// LS Electric XG5000 project: 동남138
// PLC NewPLC
// module base 0 slot 0: 입출력 모듈:XBC-DN/DP14E (DC 24V 입력 8점, 트랜지스터 출력 6점)

PROGRAM NewProgram (task: 스캔 프로그램)

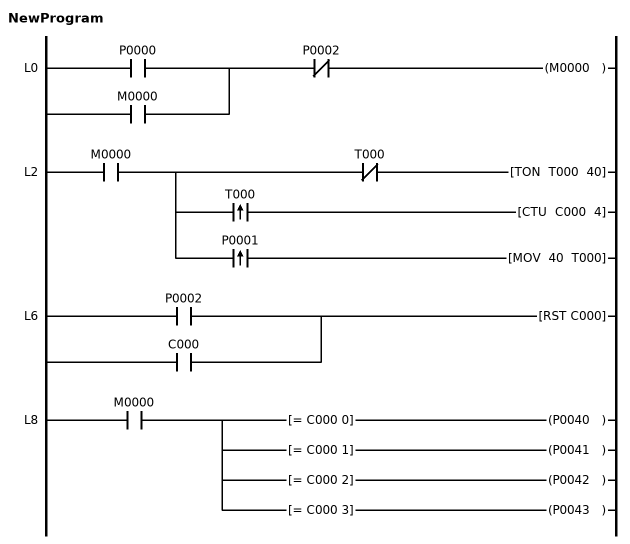
; L0
LOAD      P0000
OR        M0000
AND NOT   P0002
OUT       M0000
; L2
LOAD      M0000
MPUSH
AND NOT   T000
TON       T000 40
MLOAD
ANDP      T000
CTU       C000 4
MPOP
ANDP      P0001
MOV       40 T000
; L6
LOAD      P0002
OR        C000
RST       C000
; L8
LOAD      M0000
MPUSH
AND=      C000 0
OUT       P0040
MLOAD
AND=      C000 1
OUT       P0041
MLOAD
AND=      C000 2
OUT       P0042
MPOP
AND=      C000 3
OUT       P0043